(* PLC project CoDeSys External Library Template, WAGO e!COCKPIT e!COCKPIT, author 3S - Smart Software Solutions GmbH *)
(* stored: creationDateTime 2019-10-29T12:22:40.3755581, version 3.5.5.30, modificationDateTime 2019-10-24T14:40:07.960949, organization 3S - Smart Software Solutions GmbH *)
(* Library project template with all possible element types, docu and a sample project structure *)

(* values of enumPPPSFriskoATTOM1SErrorKlasa: AlarmCzujnikaZewnetrznego: alarm braku zmiany wartości czujnika temp. zewnetrznj; AlarmCzujnikaZasilaniaObwoduCO: alarm braku zmiany wartości czujnika temp. zasilana obwod c. o.; BrakOsiagnieciaTemperaturyCO: alarm braku osiągnięcia temp. zadanej obwodu c. o.; BladIloscPomiarowTemperatury: alarm zbyt małej ilości pomiarów dokonanych w ciągu dnia do obliczenia średniej *)

(* Autor: Paweł Kąkol, 2018-09-03-PK Prawa majątkowe: Solwena Sp. z o.o., Aktualizacje: 2019-02-19-AWy: dodanie alarmów czujnika zew., zasilania c.o., braku osiągnięcia temperatury zadanej 2019-02-18-AWy: zmiana klas alarmów Opis: enum służy do definicji klas alarmów w fb węzła Climatix POL63x na budynkach PPP Sopot (ENGIE) *)
{attribute 'qualified_only'}
{attribute 'strict'}
TYPE enumPPPSFriskoATTOM1SErrorKlasa : (BrakKomunikacji := enumKlasaAlarmu.AwariaAutomatyki, AlarmCzujnikaZewnetrznego := enumKlasaAlarmu.AwariaAutomatyki, AlarmCzujnikaZasilaniaObwoduCO := enumKlasaAlarmu.AwariaAutomatyki, BrakOsiagnieciaTemperaturyCO := enumKlasaAlarmu.Ostrzezenie, BladIloscPomiarowTemperatury := enumKlasaAlarmu.AwariaAutomatyki);
END_TYPE
